(* PLC project Sin nombre, Desconocido Sin nombre 1 *)
(* stored: creationDateTime 2025-07-13T20:27:28, modificationDateTime 2025-07-13T22:11:13 *)

PROGRAM semaforo
  VAR
    rojoc : BOOL;  (* Luz roja para carros *)
    amarillo : BOOL;  (* Luz amarilla para carros *)
    verdec : BOOL;  (* Luz verde para carros *)
    rojop : BOOL;  (* Luz roja para peatones *)
    verdep : BOOL;  (* Luz verde para peatones *)
    cont1 : BOOL;  (* Contactor 1 *)
    cont2 : BOOL;  (* Contactor 2 *)
    parada : BOOL;  (* Solicitud de parada por el usuario *)
    detener : BOOL;  (* Sostener parada *)
    cambio : BOOL;  (* Solicitud de via por el peaton *)
    conmutar : BOOL;  (* Sostener solicitud de via por el peaton *)
    T1 : BOOL;  (* Estado 1 - de rojo a verde *)
    T2 : BOOL;  (* Estado 2 - verde *)
    T3 : BOOL;  (* Estado 3 - de verde a rojo *)
    T3aux1 : BOOL;  (* Estado Aux 1 - de verde a rojo *)
    T3aux2 : BOOL;  (* Estado Aux 2 - de verde a rojo *)
    TON0 : TON;  (* Temporizador para segunda secuencia de salida *)
    TON1 : TON;  (* Temporizador para tercera secuencia de salida *)
    TON2 : TON;  (* Temporizador para cuarta secuencia de salida *)
    TON3 : TON;  (* Temporizador auxiliar para cuarta secuencia de salida *)
    TON4 : TON;  (* Temporizador de reinicio *)
    reboot : BOOL;  (* Reiniciar ciclo *)
  END_VAR

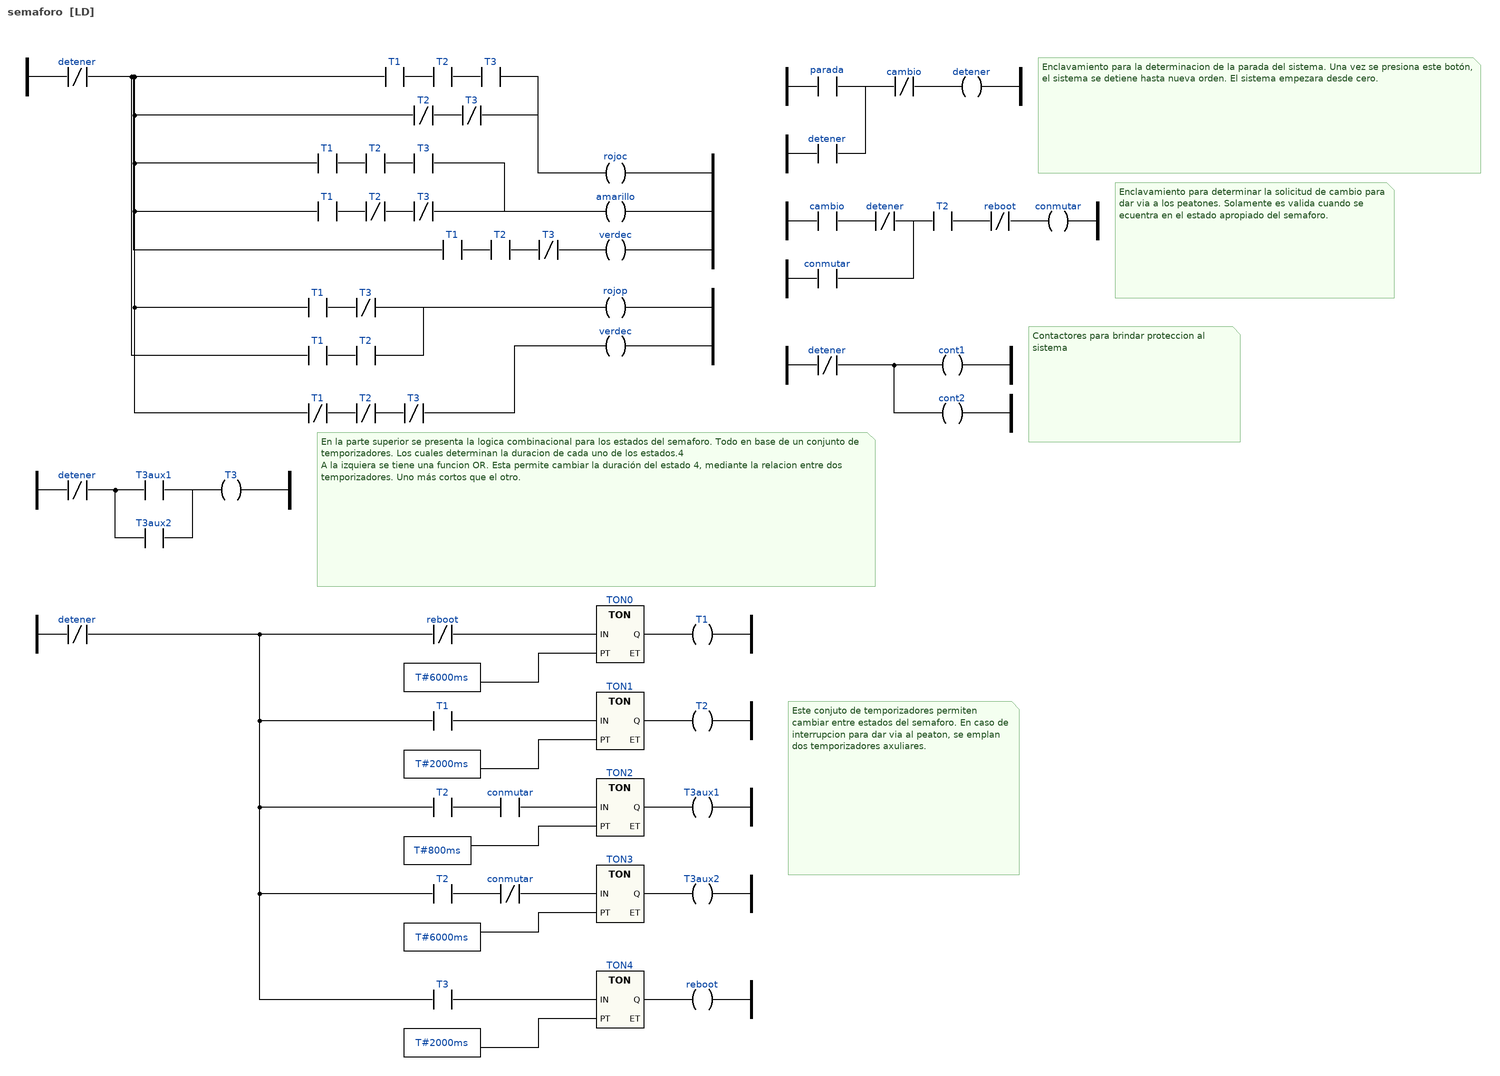
(* LD diagram, written out as Structured Text *)
(* Enclavamiento para la determinacion de la parada del sistema. Una vez se presiona este botón, el sistema se detiene hasta nueva orden. El sistema empezara desde cero. *)
rojoc := NOT detener AND (NOT T2 AND NOT T3 OR T1 AND T2 AND T3);
(* Enclavamiento para determinar la solicitud de cambio para dar via a los peatones. Solamente es valida cuando se ecuentra en el estado apropiado del semaforo. *)
amarillo := NOT detener AND T1 AND (NOT T2 AND NOT T3 OR T2 AND T3);
verdec := NOT detener AND T1 AND T2 AND NOT T3;
rojop := NOT detener AND T1 AND (NOT T3 OR T2);
(* Contactores para brindar proteccion al sistema *)
verdec := NOT detener AND NOT T1 AND NOT T2 AND NOT T3;
(* En la parte superior se presenta la logica combinacional para los estados del semaforo. Todo en base de un conjunto de temporizadores. Los cuales determinan la duracion de cada uno de los estados.4
A la izquiera se tiene una funcion OR. Esta permite cambiar la duración del estado 4, mediante la relacion entre dos temporizadores. Uno más cortos que el otro. *)
TON0(IN := NOT detener AND NOT reboot, PT := T#6000ms);
T1 := TON0.Q;
(* Este conjuto de temporizadores permiten cambiar entre estados del semaforo. En caso de interrupcion para dar via al peaton, se emplan dos temporizadores axuliares. *)
TON1(IN := NOT detener AND T1, PT := T#2000ms);
T2 := TON1.Q;
TON3(IN := NOT detener AND T2 AND NOT conmutar, PT := T#6000ms);
T3aux2 := TON3.Q;
TON2(IN := NOT detener AND T2 AND conmutar, PT := T#800ms);
T3aux1 := TON2.Q;
T3 := NOT detener AND (T3aux1 OR T3aux2);
TON4(IN := NOT detener AND T3, PT := T#2000ms);
reboot := TON4.Q;
detener := (detener OR parada) AND NOT cambio;
conmutar := (cambio AND NOT detener OR conmutar) AND T2 AND NOT reboot;
cont1 := NOT detener;
cont2 := NOT detener;
END_PROGRAM

CONFIGURATION Config0
  RESOURCE Res0 ON PLC
    TASK task0(INTERVAL := T#20ms, PRIORITY := 0);
    PROGRAM instance0 WITH task0 : semaforo;
  END_RESOURCE
END_CONFIGURATION
